SUBAPPLICATION Uebung_029 (* LED_DO Blinkende LED *)
  (* Standard: 61499-2; Description: Copyright (c) 2023 Meisterschulen am Ostbahnhof This program and the accompanying materials are made available under the terms of the Eclipse Public License 2.0 which is available at https://www.eclipse.org/legal/epl-2.0/ SPDX-License-Identifier: EPL-2.0 *)
  (* Version 1.0, 2023-10-23, Franz Höpfinger, Meisterschulen am Ostbahnhof, initial API and implementation and/or initial documentation *)
  PACKAGE Uebungen;
  IMPORT logiBUS::io::DI::logiBUS_DI::Input_I1;
  IMPORT logiBUS::io::DI::logiBUS_DI::Input_I2;
  IMPORT logiBUS::io::DI::logiBUS_DI::Input_I3;
  IMPORT logiBUS::io::DO_LED::LED_FREQ;
  IMPORT logiBUS::io::DQ::logiBUS_DO::Output_Q1;
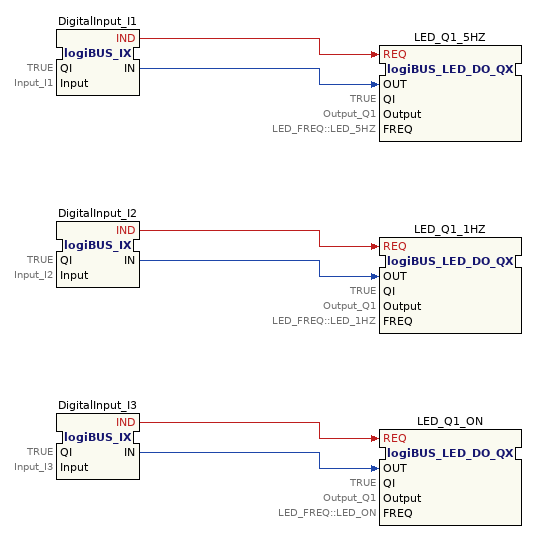
  FBS
    LED_Q1_5HZ : logiBUS::io::DO_LED::logiBUS_LED_DO_QX(QI := TRUE, Output := Output_Q1, FREQ := LED_FREQ::LED_5HZ);
    DigitalInput_I1 : logiBUS::io::DI::logiBUS_IX(QI := TRUE, Input := Input_I1);
    LED_Q1_1HZ : logiBUS::io::DO_LED::logiBUS_LED_DO_QX(QI := TRUE, Output := Output_Q1, FREQ := LED_FREQ::LED_1HZ);
    DigitalInput_I2 : logiBUS::io::DI::logiBUS_IX(QI := TRUE, Input := Input_I2);
    LED_Q1_ON : logiBUS::io::DO_LED::logiBUS_LED_DO_QX(QI := TRUE, Output := Output_Q1, FREQ := LED_FREQ::LED_ON);
    DigitalInput_I3 : logiBUS::io::DI::logiBUS_IX(QI := TRUE, Input := Input_I3);
  END_FBS
  EVENT_CONNECTIONS
    DigitalInput_I1.IND TO LED_Q1_5HZ.REQ;
    DigitalInput_I2.IND TO LED_Q1_1HZ.REQ;
    DigitalInput_I3.IND TO LED_Q1_ON.REQ;
  END_CONNECTIONS
  DATA_CONNECTIONS
    DigitalInput_I1.IN TO LED_Q1_5HZ.OUT;
    DigitalInput_I2.IN TO LED_Q1_1HZ.OUT;
    DigitalInput_I3.IN TO LED_Q1_ON.OUT;
  END_CONNECTIONS
END_SUBAPPLICATION
